// Mitsubishi GX Works2 project: theory2   PLC: FX3G

// global labels: Global1
VAR_GLOBAL
  New_Pack AT X010 : BOOL;
  Sen_Reverse AT X001 : BOOL;
  Sen_Forward AT X002 : BOOL;
  Timer_Unload_finish AT TS0 : BOOL;
  Light_Forward AT Y000 : BOOL;
  Light_Reverse AT Y001 : BOOL;
  Timer_Unload_counter AT TC0 : BOOL;
END_VAR
VAR_GLOBAL CONSTANT
  Unload_time : INT := 150;
END_VAR
VAR_GLOBAL
  light_timer AT Y011 : BOOL;
END_VAR

// task Task_01 (event TRUE, interval 0, priority 31): POU_01

PROGRAM POU_01
(* structured ladder/FBD written out as ST: instructions are called as NAME(EN, inputs, outputs); _pN, _eN, _tN stand for wires *)
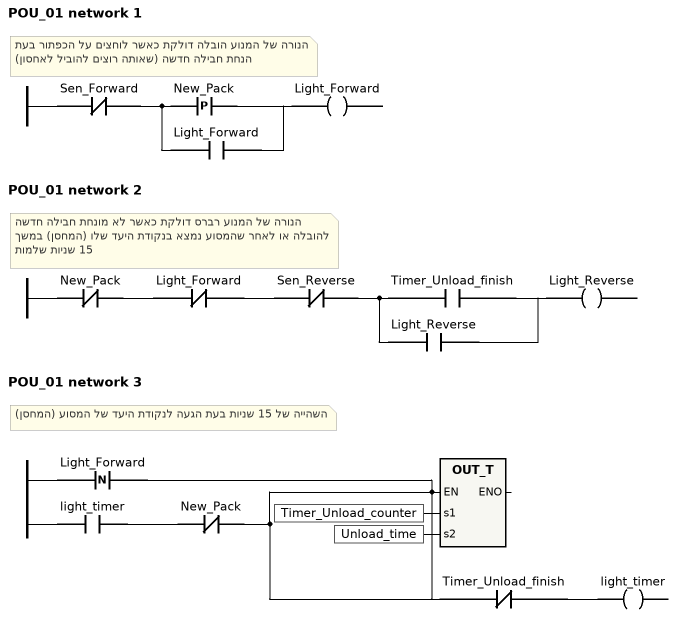
(* network 1 *)
(* הנורה של המנוע הובלה דולקת כאשר לוחצים על הכפתור בעת הנחת חבילה חדשה (שאותה רוצים להוביל לאחסון) *)
_p1 := NOT Sen_Forward;
Light_Forward := (_p1 AND LDP(TRUE, New_Pack)) OR (_p1 AND Light_Forward);
(* network 2 *)
(* הנורה של המנוע רברס דולקת כאשר לא מונחת חבילה חדשה להובלה או לאחר שהמסוע נמצא בנקודת היעד שלו (המחסן) במשך 15 שניות שלמות *)
_p1 := NOT New_Pack AND NOT Light_Forward AND NOT Sen_Reverse;
Light_Reverse := (_p1 AND Timer_Unload_finish) OR (_p1 AND Light_Reverse);
(* network 3 *)
(* השהייה של 15 שניות בעת הגעה לנקודת היעד של המסוע (המחסן) *)
_p1 := LDF(TRUE, Light_Forward) OR (light_timer AND NOT New_Pack);
light_timer := _p1 AND NOT Timer_Unload_finish;
OUT_T(_p1, Timer_Unload_counter, Unload_time);
END_PROGRAM
